// TIA Portal project "WaterTankControl1" (V20)

(* hardware
DEVICE "S7-1500/ET200MP station_1"  S7-1500 station
   slot 0: "Rail_0"  Rack  6ES7 590-1***0-0AA0
   slot 1: "PLC_1"  CPU 1511-1 PN  6ES7 511-1AL03-0AB0  V4.0
      slot 3: "CPU display_1"  6ES7591-1AA00-0AA0
      slot 32768: "PROFINET interface_1"  X1
         slot 32769: "Port_1"  X1 P1
         slot 32770: "Port_2"  X1 P2
      slot 34817: "Virtual CP interface port_1"  Virtual CP interface port  Virtual CP interface port FW V4.0
*)

// ===== PLC "PLC_1"  CPU 1511-1 PN =====

VAR_GLOBAL   // PLC tag table "Default tag table"
   "LevelLow" AT %I0.0 : Bool;
   "LevelMedium" AT %I0.1 : Bool;
   "LevelHigh" AT %I0.2 : Bool;
   "StartBtn" AT %I0.3 : Bool;
   "StopBtn" AT %I0.4 : Bool;
   "EStop" AT %I0.5 : Bool;
   "LevelRaw" AT %IW64 : Int;
   "InletValve" AT %Q0.0 : Bool;
   "OutletPump" AT %Q0.1 : Bool;
   "AlarmOverflow" AT %Q0.2 : Bool;
   "AlarmDryRun" AT %Q0.3 : Bool;
   "SystemRunning" AT %Q0.4 : Bool;
END_VAR

DATA_BLOCK "TankData"   // DB1
{ S7_Optimized_Access := 'TRUE' }
VERSION : 0.1
   VAR
      LevelRaw : Int := 0;   // Raw analog input 0 to 27648
      LevelPercent : Real;   // Scaled level 0 to 100 percent
      InletValve : Bool;   // Inlet valve command status
      OutletPump : Bool;   // Outlet pump command status
      SystemRunning : Bool;   // System run status
      AlarmOverflow : Bool;   // Overflow alarm active
      AlarmDryRun : Bool;   // Dry run alarm active
      FillRate : Real;   // Fill rate percent per minute
      DrainRate : Real;   // Drain rate percent per minute
      AITimeToEmpty : Real := 999.0;   // AI prediction minutes until empty
      CycleCount : Int;   // Number of completed fill cycles
   END_VAR
BEGIN
END_DATA_BLOCK

DATA_BLOCK "TankControl_DB"   // DB2
{ S7_Optimized_Access := 'TRUE' }
VERSION : 0.1
// stored: InstanceOfName TankControl
"TankControl"
BEGIN
END_DATA_BLOCK

DATA_BLOCK "RateCalc_DB"   // DB3
{ S7_Optimized_Access := 'TRUE' }
VERSION : 0.1
// stored: InstanceOfName RateCalc
"RateCalc"
BEGIN
END_DATA_BLOCK

FUNCTION_BLOCK "TankControl"   // FB1, SCL
{ S7_Optimized_Access := 'TRUE' }
VERSION : 0.1
   VAR_INPUT
      StartBtn : Bool;
      StopBtn : Bool;
      EStop : Bool;
      LevelLow : Bool;
      LevelMedium : Bool;
      LevelHigh : Bool;
      LevelPercent : Real;
   END_VAR
   VAR_OUTPUT
      InletValve : Bool;
      OutletPump : Bool;
      AlarmOverflow : Bool;
      AlarmDryRun : Bool;
      SystemRunning : Bool;
   END_VAR
   VAR
      RunLatch : Bool;
      ValveLatch : Bool;
   END_VAR
BEGIN
   IF #EStop THEN
       #RunLatch := FALSE;
       #ValveLatch := FALSE;
       #InletValve := FALSE;
       #OutletPump := FALSE;
       #AlarmOverflow := FALSE;
       #AlarmDryRun := FALSE;
       #SystemRunning := FALSE;
       RETURN;
   END_IF;

   IF #StartBtn THEN
       #RunLatch := TRUE;
   END_IF;

   IF #StopBtn THEN
       #RunLatch := FALSE;
       #ValveLatch := FALSE;
   END_IF;

   #SystemRunning := #RunLatch;

   IF #RunLatch THEN

       #OutletPump := TRUE;

       IF #LevelLow THEN
           #ValveLatch := TRUE;
       END_IF;

       IF #LevelHigh THEN
           #ValveLatch := FALSE;
       END_IF;

       #InletValve := #ValveLatch;

       IF #LevelPercent > REAL#95.0 THEN
           IF #InletValve THEN
               #AlarmOverflow := TRUE;
               #InletValve := FALSE;
               #ValveLatch := FALSE;
           END_IF;
       ELSE
           #AlarmOverflow := FALSE;
       END_IF;

       IF #LevelPercent < REAL#5.0 THEN
           IF #OutletPump THEN
               #AlarmDryRun := TRUE;
               #OutletPump := FALSE;
           END_IF;
       ELSE
           #AlarmDryRun := FALSE;
       END_IF;

   ELSE
       #InletValve := FALSE;
       #OutletPump := FALSE;

   END_IF;
END_FUNCTION_BLOCK

FUNCTION_BLOCK "RateCalc"   // FB2, SCL
{ S7_Optimized_Access := 'TRUE' }
VERSION : 0.1
   VAR_INPUT
      CurrentLevel : Real;
      InletValve : Bool;
      OutletPump : Bool;
   END_VAR
   VAR_OUTPUT
      FillRate : Real;
      DrainRate : Real;
   END_VAR
   VAR
      PrevLevel : Real;
      SampleTimer : TON_TIME;
   END_VAR
BEGIN
   // ════════════════════════════════════════════════
   // FB2 — RateCalc
   // Measures fill and drain rate in percent/minute
   // Samples level every 10 seconds for stable result
   // ════════════════════════════════════════════════

   // ── Start the 10 second timer ─────────────────
   // WHY: TON counts time. IN=TRUE starts counting.
   // PT=T#10S sets the target to 10 seconds.
   // Q goes TRUE when 10 seconds have elapsed.
   // Timer resets when IN goes FALSE.

   #SampleTimer(IN := TRUE,
                PT := T#10S);

   // ── Only calculate when 10 seconds elapsed ─────
   IF #SampleTimer.Q THEN

       // How much did level change in last 10 seconds?
       // Positive number = filling
       // Negative number = draining
       IF (#CurrentLevel - #PrevLevel) > REAL#0.0 THEN
           // Tank is filling
           // Multiply by 6 converts per-10s to per-minute
           // WHY 6: 60 seconds / 10 seconds = 6 samples per minute
           #FillRate := (#CurrentLevel - #PrevLevel) * REAL#6.0;
       END_IF;

       IF (#CurrentLevel - #PrevLevel) < REAL#0.0 THEN
           // Tank is draining
           // Difference is negative so multiply by -6
           // to get a positive drain rate value
           #DrainRate := (#PrevLevel - #CurrentLevel) * REAL#6.0;
       END_IF;

       // Store current level for next calculation
       #PrevLevel := #CurrentLevel;

       // Reset timer so it starts counting again
       // WHY: Setting IN=FALSE resets the TON timer
       // Next scan IN goes TRUE again and counting restarts
       #SampleTimer(IN := FALSE,
                    PT := T#10S);

   END_IF;
END_FUNCTION_BLOCK

FUNCTION "ScaleLevel" : Real   // FC1, SCL
{ S7_Optimized_Access := 'TRUE' }
VERSION : 0.1
   VAR_INPUT
      RawValue : Int;
      ScaleMin : Real;
      ScaleMax : Real;
   END_VAR
BEGIN
   // ══════════════════════════════════════════
   // FC1 — ScaleLevel
   // Converts raw analog (0-27648) to 0-100%
   // ══════════════════════════════════════════

   // Calculate scaled value
   // INT_TO_REAL converts integer to decimal number
   // so division works correctly
   #ScaleLevel := ((INT_TO_REAL(#RawValue) / 27648.0) * (#ScaleMax - #ScaleMin)) + #ScaleMin;

   // Clamp — never return value outside valid range
   IF #ScaleLevel > #ScaleMax THEN
       #ScaleLevel := #ScaleMax;
   ELSIF #ScaleLevel < #ScaleMin THEN
       #ScaleLevel := #ScaleMin;
   END_IF;
END_FUNCTION

ORGANIZATION_BLOCK "Main"   // OB1, SCL, ProgramCycle
TITLE = "Main Program Sweep (Cycle)"
{ S7_Optimized_Access := 'TRUE' }
VERSION : 0.1
   VAR_INPUT
      Initial_Call : Bool;   // Initial call of this OB
      Remanence : Bool;   // =True, if remanent data are available
   END_VAR
BEGIN
   "TankData".LevelRaw := "LevelRaw";

   "TankData".LevelPercent := "ScaleLevel"(
                                           RawValue := "TankData".LevelRaw,
                                           ScaleMin := REAL#0.0,
                                           ScaleMax := REAL#100.0
   );

   "TankControl_DB"(
                    StartBtn      := "StartBtn",
                    StopBtn       := "StopBtn",
                    EStop         := "EStop",
                    LevelLow      := "LevelLow",
                    LevelMedium   := "LevelMedium",
                    LevelHigh     := "LevelHigh",
                    LevelPercent  := "TankData".LevelPercent
   );

   "TankData".InletValve := "TankControl_DB".InletValve;
   "TankData".OutletPump := "TankControl_DB".OutletPump;
   "TankData".AlarmOverflow := "TankControl_DB".AlarmOverflow;
   "TankData".AlarmDryRun := "TankControl_DB".AlarmDryRun;
   "TankData".SystemRunning := "TankControl_DB".SystemRunning;

   "RateCalc_DB"(
                 CurrentLevel := "TankData".LevelPercent,
                 InletValve   := "TankData".InletValve,
                 OutletPump   := "TankData".OutletPump
   );

   "TankData".FillRate := "RateCalc_DB".FillRate;
   "TankData".DrainRate := "RateCalc_DB".DrainRate;

   "InletValve" := "TankData".InletValve;
   "OutletPump" := "TankData".OutletPump;
   "AlarmOverflow" := "TankData".AlarmOverflow;
   "AlarmDryRun" := "TankData".AlarmDryRun;
   "SystemRunning" := "TankData".SystemRunning;
END_ORGANIZATION_BLOCK